Fanuc TP program (LS listing): ls_test.ls

/PROG  LS_TEST
/ATTR
OWNER		= MNEDITOR;
COMMENT		= "";
PROG_SIZE	= 279;
CREATE		= DATE 21-08-19  TIME 21:16:00;
MODIFIED	= DATE 21-08-19  TIME 21:16:00;
FILE_NAME	= ;
VERSION		= 0;
LINE_COUNT	= 5;
MEMORY_SIZE	= 631;
PROTECT		= READ_WRITE;
TCD:  STACK_SIZE	= 0,
      TASK_PRIORITY	= 50,
      TIME_SLICE	= 0,
      BUSY_LAMP_OFF	= 0,
      ABORT_REQUEST	= 0,
      PAUSE_REQUEST	= 0;
DEFAULT_GROUP	= 1,*,*,*,*;
CONTROL_CODE	= 00000000 00000000;
/APPL
/APPL

AUTO_SINGULARITY_HEADER;
  ENABLE_SINGULARITY_AVOIDANCE   : TRUE;
/MN
   1:  !One Comment started*** ;
   2:   ;
   3:  !Added Comment from Vs ;
   4:   ;
   5:  !This line added out of order ;
/POS
/END
